FUNCTION_BLOCK HASHTBL (* Service Interface to java.util.Hashtable *)
  (* Standard: 61499 Feasibility Demo ITA *)
  (* Version 0.1, 2000-04-21, JHC, Rockwell Automation, Re-implemented *)
  (* Compiler header: package fb.rt.math; import java.util.*; *)
  (* Compiler Java IBM VisualAge 3.0 *)
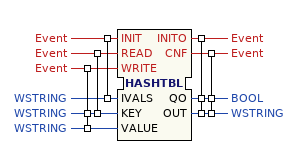
  EVENT_INPUT
    INIT WITH IVALS; (* Clear/Initialize Table *)
    READ WITH KEY; (* Read the Value Corresponding to a Key *)
    WRITE WITH KEY, VALUE; (* Record the Value Corresponding to a Key *)
  END_EVENT
  EVENT_OUTPUT
    INITO WITH QO, OUT; (* Initialization Confirm,OUT=Empty *)
    CNF WITH QO, OUT; (* READ/WRITE Result *)
  END_EVENT
  VAR_INPUT
    IVALS : WSTRING; (* KEY/VALUE Pairs,Comma-Separated *)
    KEY : WSTRING; (* READ/WRITE Key *)
    VALUE : WSTRING; (* WRITE value *)
  END_VAR
  VAR_OUTPUT
    QO : BOOL; (* 0=No Match Found *)
    OUT : WSTRING; (* READ/WRITE result *)
  END_VAR
  SERVICE APPLICATION/Hashtable
    SEQUENCE init_table
      APPLICATION.INIT(KEYS,VALUES) -> Hashtable.clear() -> APPLICATION.INITO+(OUT);
    END_SEQUENCE
    SEQUENCE normal_read (* OUT=VALUE Matching KEY *)
      APPLICATION.READ(KEY) -> Hashtable.get(KEY) -> APPLICATION.CNF+(OUT);
    END_SEQUENCE
    SEQUENCE read_no_match (* No match for KEY,OUT=Empty String *)
      APPLICATION.READ(KEY) -> Hashtable.get(KEY) -> APPLICATION.CNF-("");
    END_SEQUENCE
    SEQUENCE write (* OUT=VALUE *)
      APPLICATION.WRITE(KEY,VALUE) -> Hashtable.put(KEY,VALUE) -> APPLICATION.CNF+(OUT);
    END_SEQUENCE
  END_SERVICE
END_FUNCTION_BLOCK
